Staubli VAL3: markListAdd.pgx

program markListAdd(string x_sEvent)
begin
  // add in the queue
  if sMarkList!=""
    insert(sMarkList[size(sMarkList)])
  endIf
  sMarkList[size(sMarkList)-1]=x_sEvent
end
